{attribute 'GeneratedUsingTerminal: EK1122-0000-0018'}
{attribute addProperty BoxType "EK1122-0000-0018"}
{attribute addProperty Id "Drive_A20_CMMT_ASCMMT_F160324F49Drive_A21_CMMT_ASCMMT_ABED948241"}
{attribute addProperty CRC "4258478301"}
{attribute addProperty Size "90"}
TYPE Term_146_EK1122_FDD338DD EXTENDS EK1122_1FC0878B :
STRUCT
	{attribute addProperty Name "Drive_A20_CMMT_AS"}
	{attribute addProperty PreviousPort "Term 146 (EK1122) : D"}
	Drive_A20_CMMT_AS : CMMT_F160324F;
	{attribute addProperty Name "Drive_A21_CMMT_AS"}
	{attribute addProperty PreviousPort "Drive A20 (CMMT-AS) : B"}
	Drive_A21_CMMT_AS : CMMT_ABED9482;
END_STRUCT
END_TYPE

(* stored: Version 1.2.0.0, ProductVersion 3.1.4024.9
   DUT Term_146_EK1122_FDD338DD: Id {a0ba6d7a-3acc-0f28-0eb7-1637380090dc} *)
